(*
SPDX-FileCopyrightText: © 2026 Oleksandr Tiutyk <trofimich@gmail.com>
SPDX-License-Identifier: MIT
License: https://opensource.org/license/mit
*)

(*!
<summary>Defines a condition that compares a named variable against a configured reference value.</summary>
<description>
Standard elements resolve condition-local and ancestor bindings first, then evaluating activity/ancestor
bindings, then workflow fallback. The condition-associated workflow precedes a distinct context workflow.
Custom elements expose direct bindings through ILocalVariableLookup; legacy opaque lookups run after
discoverable local scopes and before workflow fallback.
</description>
*)

INTERFACE IVariableHasValueCondition EXTENDS ICondition

(*!
<summary>Configures the monitored variable name and copies the reference value for comparison.</summary>
<param name="monitoredVariableName">Non-empty name of the variable to look up during evaluation.</param>
<param name="referenceValue">Non-empty reference value to compare against.</param>
*)
METHOD Configure
VAR_INPUT
	monitoredVariableName : STRING;
	referenceValue : ANY; 
END_VAR
END_METHOD

(*!
<summary>Returns the configured variable name.</summary>
*)
{attribute 'monitoring' := 'call'}
PROPERTY MonitoredVariableName : STRING
GET
END_GET
END_PROPERTY

(*!
<summary>Returns a borrowed reference to the stored comparison value.</summary>
*)
{attribute 'monitoring' := 'call'}
PROPERTY ReferenceValue : REFERENCE TO TOF_Core.GENERIC_VALUE
GET
END_GET
END_PROPERTY

END_INTERFACE

(* stored: Version 1.1.0.1
   Itf IVariableHasValueCondition: Id {f41d5a3f-0b80-4e3d-84ca-b11d606174d2}
   Method Configure: Id {ca8f5004-2674-4419-ba89-4d26be48f8b5}
   Property MonitoredVariableName: Id {147107e1-9526-4e67-ab32-cb4812acd99e}
   Get Get: Id {f20cd9c8-6aee-4d61-8420-ad95e40523c2}
   Property ReferenceValue: Id {d2daa20e-c057-41c3-b95c-c3195de25cd8}
   Get Get: Id {285ee67d-c572-43e8-ab14-fc782d1497ea} *)
